// TIA Portal project "LECTOR CODIGO DE BARRAS" (V11)

(* hardware
DEVICE "S7300/ET200 station_1"  SIMATIC 300-Station
   slot 0: "Perfil soporte_0"  Rail  6ES7 390-1***0-0AA0
   slot 2: "PLC_1"  CPU 313C-2 DP  6ES7 313-6CF03-0AB0  V2.6
      slot 0: "Interfaz MPI_1"  MPI
      slot 1: "Interfaz DP_1"  DP
      slot 2: "DI16/DO16_1"  DI16/DO16
      slot 4: "Contaje_1"  Counter
   slot 4: "CP 343-1 Lean_1"  CP 343-1 LEAN  6GK7 343-1CX10-0XE0  V2.4
*)

// ===== PLC "PLC_1"  CPU 313C-2 DP =====

VAR_GLOBAL   // PLC tag table "Tabla de variables estándar"
   "ON PERMITE OFF NO" AT %I0.0 : Bool;
   "CANCELA LECTURA" AT %I0.1 : Bool;
   "Tag_2" AT %M0.0 : Bool;
   "Tag_4" AT %M0.1 : Bool;
   "Tag_5" AT %MW6 : Int;
   "Tag_7" AT %MW8 : Word;
   "Tag_1" AT %MW10 : Int;
   "Tag_3" AT %MD12 : Real;
   "Tag_6" AT %MW16 : Int;
   "Tag_14" AT %MD18 : Real;
   "Tag_15" AT %MW22 : Int;
   "Tag_16" AT %MD24 : Real;
   "Tag_17" AT %MW28 : Int;
   "Tag_18" AT %MD30 : Real;
   "Tag_19" AT %MD34 : Real;
   "Tag_20" AT %MD40 : Real;
   "RECTIFICAR FACTURA" AT %I0.2 : Bool;
   "RESET" AT %I0.3 : Bool;
   "Tag_8" AT %I0.4 : Bool;
   "Tag_9" AT %I0.5 : Bool;
   "Tag_10" AT %I0.6 : Bool;
   "Tag_11" AT %I0.7 : Bool;
   "Tag_12" AT %I1.0 : Bool;
   "Tag_13" AT %I1.1 : Bool;
   "Tag_21" AT %I1.2 : Bool;
   "Tag_22" AT %I1.3 : Bool;
   "Tag_23" AT %I1.4 : Bool;
   "Tag_24" AT %I1.5 : Bool;
   "Tag_25" AT %Q0.0 : Bool;
   "Tag_26" AT %Q0.1 : Bool;
   "Tag_27" AT %Q0.2 : Bool;
   "Tag_28" AT %Q0.3 : Bool;
   "Tag_29" AT %Q0.4 : Bool;
   "Tag_30" AT %I1.6 : Bool;
END_VAR

DATA_BLOCK "CODIGO CAMEL"   // DB1
{ S7_Optimized_Access := 'FALSE' }
VERSION : 0.1
   VAR
      CAMEL : Array [0..20] of Byte;
   END_VAR
BEGIN
   CAMEL[0] := '8';
   CAMEL[1] := '4';
   CAMEL[2] := '1';
   CAMEL[3] := '6';
   CAMEL[4] := '5';
   CAMEL[5] := '9';
   CAMEL[6] := '6';
   CAMEL[7] := '1';
END_DATA_BLOCK

DATA_BLOCK "CODIGO PALL MALL"   // DB2
{ S7_Optimized_Access := 'FALSE' }
VERSION : 0.1
   VAR
      "PALL MALL" : Array [0..20] of Byte;
   END_VAR
BEGIN
   "PALL MALL"[0] := '8';
   "PALL MALL"[1] := '4';
   "PALL MALL"[2] := '1';
   "PALL MALL"[3] := '6';
   "PALL MALL"[4] := '0';
   "PALL MALL"[5] := '9';
   "PALL MALL"[6] := '6';
   "PALL MALL"[7] := '6';
END_DATA_BLOCK

DATA_BLOCK "CODIGO FORTUNA"   // DB3
{ S7_Optimized_Access := 'FALSE' }
VERSION : 0.1
   VAR
      FORTUNA : Array [0..20] of Byte;
   END_VAR
BEGIN
   FORTUNA[0] := '8';
   FORTUNA[1] := '4';
   FORTUNA[2] := '1';
   FORTUNA[3] := '6';
   FORTUNA[4] := '0';
   FORTUNA[5] := '0';
   FORTUNA[6] := '2';
   FORTUNA[7] := '7';
END_DATA_BLOCK

DATA_BLOCK "LECTURA LECTOR"   // DB4
{ S7_Optimized_Access := 'FALSE' }
VERSION : 0.1
   VAR
      "LECTURA LECTOR" : Array [0..20] of Byte;
   END_VAR
BEGIN
END_DATA_BLOCK

DATA_BLOCK "CODIGO LUCKY"   // DB6
{ S7_Optimized_Access := 'FALSE' }
VERSION : 0.1
   VAR
      "CODIGO LUCKY" : Array [0..20] of Byte;
   END_VAR
BEGIN
   "CODIGO LUCKY"[0] := '8';
   "CODIGO LUCKY"[1] := '4';
   "CODIGO LUCKY"[2] := '1';
   "CODIGO LUCKY"[3] := '6';
   "CODIGO LUCKY"[4] := '0';
   "CODIGO LUCKY"[5] := '0';
   "CODIGO LUCKY"[6] := '8';
   "CODIGO LUCKY"[7] := '9';
END_DATA_BLOCK

DATA_BLOCK "DATOS AUXILIARES"   // DB7
{ S7_Optimized_Access := 'FALSE' }
VERSION : 0.1
   VAR
      DATOS : Array [0..41] of Bool;
      "CONTADOR UNID." : Array [0..3] of Int;
      "CONTADOR PVP TOTAL" : Array [0..3] of Real;
      "CONTADOR FACTURA TOTAL" : Array [0..0] of Real;
      "BOBINAS AUX." : Array [0..8] of Bool;
   END_VAR
BEGIN
END_DATA_BLOCK

FUNCTION "REGISTRO PALL MALL." : Void   // FC1, LAD
{ S7_Optimized_Access := 'FALSE' }
VERSION : 0.1
   VAR_OUTPUT
      "UNIDADES PALL MALL" : Int;
      "P.V.P. TOTAL" : Real;
   END_VAR
   VAR_TEMP   // added for the SCL form of the ladder/FBD networks
      _w1 : Bool;
      _w2 : Bool;
   END_VAR
BEGIN

REGION Network 1
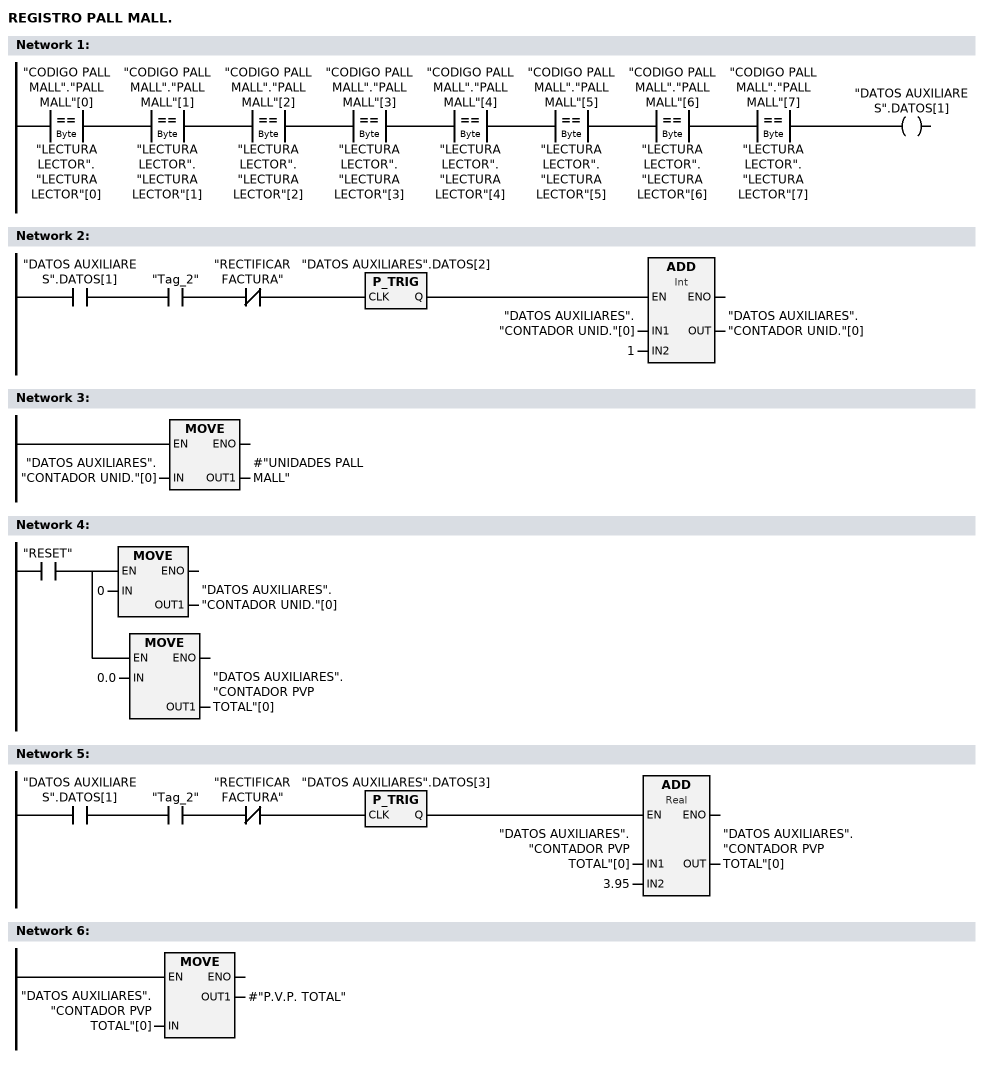
   RUNG wire#powerrail
      { S7_Templates := "SrcType := Byte" } EQ_Contact(in1 := "CODIGO PALL MALL"."PALL MALL"[0], in2 := "LECTURA LECTOR"."LECTURA LECTOR"[0])
      { S7_Templates := "SrcType := Byte" } EQ_Contact(in1 := "CODIGO PALL MALL"."PALL MALL"[1], in2 := "LECTURA LECTOR"."LECTURA LECTOR"[1])
      { S7_Templates := "SrcType := Byte" } EQ_Contact(in1 := "CODIGO PALL MALL"."PALL MALL"[2], in2 := "LECTURA LECTOR"."LECTURA LECTOR"[2])
      { S7_Templates := "SrcType := Byte" } EQ_Contact(in1 := "CODIGO PALL MALL"."PALL MALL"[3], in2 := "LECTURA LECTOR"."LECTURA LECTOR"[3])
      { S7_Templates := "SrcType := Byte" } EQ_Contact(in1 := "CODIGO PALL MALL"."PALL MALL"[4], in2 := "LECTURA LECTOR"."LECTURA LECTOR"[4])
      { S7_Templates := "SrcType := Byte" } EQ_Contact(in1 := "CODIGO PALL MALL"."PALL MALL"[5], in2 := "LECTURA LECTOR"."LECTURA LECTOR"[5])
      { S7_Templates := "SrcType := Byte" } EQ_Contact(in1 := "CODIGO PALL MALL"."PALL MALL"[6], in2 := "LECTURA LECTOR"."LECTURA LECTOR"[6])
      { S7_Templates := "SrcType := Byte" } EQ_Contact(in1 := "CODIGO PALL MALL"."PALL MALL"[7], in2 := "LECTURA LECTOR"."LECTURA LECTOR"[7])
      Coil( "DATOS AUXILIARES".DATOS[1] )
   END_RUNG
   // the same network as SCL:
   "DATOS AUXILIARES".DATOS[1] := ("CODIGO PALL MALL"."PALL MALL"[0] = "LECTURA LECTOR"."LECTURA LECTOR"[0]) AND ("CODIGO PALL MALL"."PALL MALL"[1] = "LECTURA LECTOR"."LECTURA LECTOR"[1]) AND ("CODIGO PALL MALL"."PALL MALL"[2] = "LECTURA LECTOR"."LECTURA LECTOR"[2]) AND ("CODIGO PALL MALL"."PALL MALL"[3] = "LECTURA LECTOR"."LECTURA LECTOR"[3]) AND ("CODIGO PALL MALL"."PALL MALL"[4] = "LECTURA LECTOR"."LECTURA LECTOR"[4]) AND ("CODIGO PALL MALL"."PALL MALL"[5] = "LECTURA LECTOR"."LECTURA LECTOR"[5]) AND ("CODIGO PALL MALL"."PALL MALL"[6] = "LECTURA LECTOR"."LECTURA LECTOR"[6]) AND ("CODIGO PALL MALL"."PALL MALL"[7] = "LECTURA LECTOR"."LECTURA LECTOR"[7]);
END_REGION

REGION Network 2
   RUNG wire#powerrail
      Contact( "DATOS AUXILIARES".DATOS[1] )
      Contact( "Tag_2" )
      I_Contact( "RECTIFICAR FACTURA" )
      P_Trig( "DATOS AUXILIARES".DATOS[2] )
      { S7_Templates := "SrcType := Int"; S7_GenerateENO := "TRUE" } Add(in1 := "DATOS AUXILIARES"."CONTADOR UNID."[0], in2 := 1, out => "DATOS AUXILIARES"."CONTADOR UNID."[0])
   END_RUNG
   // the same network as SCL:
   #_w1 := "DATOS AUXILIARES".DATOS[1] AND "Tag_2" AND NOT "RECTIFICAR FACTURA";
   #_w2 := #_w1 AND NOT "DATOS AUXILIARES".DATOS[2];   // rising edge
   "DATOS AUXILIARES".DATOS[2] := #_w1;
   IF #_w2 THEN "DATOS AUXILIARES"."CONTADOR UNID."[0] := "DATOS AUXILIARES"."CONTADOR UNID."[0] + 1; END_IF;
END_REGION

REGION Network 3
   RUNG wire#powerrail
      { S7_GenerateENO := "TRUE" } Move(in := "DATOS AUXILIARES"."CONTADOR UNID."[0], out1 => #"UNIDADES PALL MALL")
   END_RUNG
   // the same network as SCL:
   #"UNIDADES PALL MALL" := "DATOS AUXILIARES"."CONTADOR UNID."[0];
END_REGION

REGION Network 4
   RUNG wire#powerrail
      Contact( "RESET" )
      wire#w1
      { S7_GenerateENO := "TRUE" } Move(in := 0, out1 => "DATOS AUXILIARES"."CONTADOR UNID."[0])
   END_RUNG
   RUNG wire#w1
      { S7_GenerateENO := "TRUE" } Move(in := 0.0, out1 => "DATOS AUXILIARES"."CONTADOR PVP TOTAL"[0])
   END_RUNG
   // the same network as SCL:
   IF "RESET" THEN
       "DATOS AUXILIARES"."CONTADOR UNID."[0] := 0;
       "DATOS AUXILIARES"."CONTADOR PVP TOTAL"[0] := 0.0;
   END_IF;
END_REGION

REGION Network 5
   RUNG wire#powerrail
      Contact( "DATOS AUXILIARES".DATOS[1] )
      Contact( "Tag_2" )
      I_Contact( "RECTIFICAR FACTURA" )
      P_Trig( "DATOS AUXILIARES".DATOS[3] )
      { S7_Templates := "SrcType := Real"; S7_GenerateENO := "TRUE" } Add(in1 := "DATOS AUXILIARES"."CONTADOR PVP TOTAL"[0], in2 := 3.95, out => "DATOS AUXILIARES"."CONTADOR PVP TOTAL"[0])
   END_RUNG
   // the same network as SCL:
   #_w1 := "DATOS AUXILIARES".DATOS[1] AND "Tag_2" AND NOT "RECTIFICAR FACTURA";
   #_w2 := #_w1 AND NOT "DATOS AUXILIARES".DATOS[3];   // rising edge
   "DATOS AUXILIARES".DATOS[3] := #_w1;
   IF #_w2 THEN
       "DATOS AUXILIARES"."CONTADOR PVP TOTAL"[0] := "DATOS AUXILIARES"."CONTADOR PVP TOTAL"[0] + 3.95;
   END_IF;
END_REGION

REGION Network 6
   RUNG wire#powerrail
      { S7_GenerateENO := "TRUE" } Move(in := "DATOS AUXILIARES"."CONTADOR PVP TOTAL"[0], out1 => #"P.V.P. TOTAL")
   END_RUNG
   // the same network as SCL:
   #"P.V.P. TOTAL" := "DATOS AUXILIARES"."CONTADOR PVP TOTAL"[0];
END_REGION
END_FUNCTION

FUNCTION "REGISTRO CAMELL" : Void   // FC2, LAD
{ S7_Optimized_Access := 'FALSE' }
VERSION : 0.1
   VAR_OUTPUT
      "UNIDADES CAMELL" : Int;
      "PVP TOTAL" : Real;
   END_VAR
   VAR_TEMP   // added for the SCL form of the ladder/FBD networks
      _w1 : Bool;
      _w2 : Bool;
   END_VAR
BEGIN

REGION Network 1
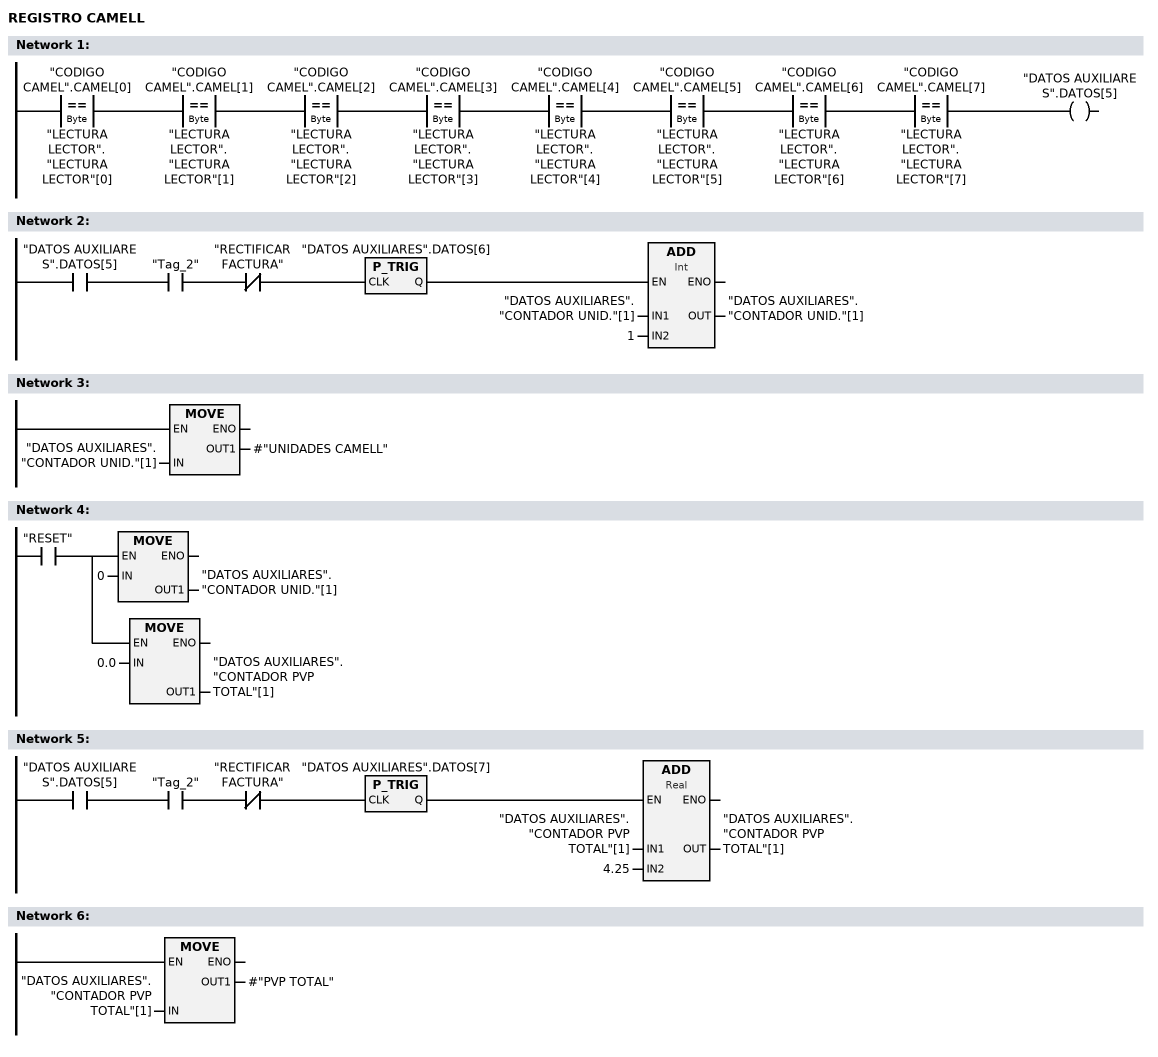
   RUNG wire#powerrail
      { S7_Templates := "SrcType := Byte" } EQ_Contact(in1 := "CODIGO CAMEL".CAMEL[0], in2 := "LECTURA LECTOR"."LECTURA LECTOR"[0])
      { S7_Templates := "SrcType := Byte" } EQ_Contact(in1 := "CODIGO CAMEL".CAMEL[1], in2 := "LECTURA LECTOR"."LECTURA LECTOR"[1])
      { S7_Templates := "SrcType := Byte" } EQ_Contact(in1 := "CODIGO CAMEL".CAMEL[2], in2 := "LECTURA LECTOR"."LECTURA LECTOR"[2])
      { S7_Templates := "SrcType := Byte" } EQ_Contact(in1 := "CODIGO CAMEL".CAMEL[3], in2 := "LECTURA LECTOR"."LECTURA LECTOR"[3])
      { S7_Templates := "SrcType := Byte" } EQ_Contact(in1 := "CODIGO CAMEL".CAMEL[4], in2 := "LECTURA LECTOR"."LECTURA LECTOR"[4])
      { S7_Templates := "SrcType := Byte" } EQ_Contact(in1 := "CODIGO CAMEL".CAMEL[5], in2 := "LECTURA LECTOR"."LECTURA LECTOR"[5])
      { S7_Templates := "SrcType := Byte" } EQ_Contact(in1 := "CODIGO CAMEL".CAMEL[6], in2 := "LECTURA LECTOR"."LECTURA LECTOR"[6])
      { S7_Templates := "SrcType := Byte" } EQ_Contact(in1 := "CODIGO CAMEL".CAMEL[7], in2 := "LECTURA LECTOR"."LECTURA LECTOR"[7])
      Coil( "DATOS AUXILIARES".DATOS[5] )
   END_RUNG
   // the same network as SCL:
   "DATOS AUXILIARES".DATOS[5] := ("CODIGO CAMEL".CAMEL[0] = "LECTURA LECTOR"."LECTURA LECTOR"[0]) AND ("CODIGO CAMEL".CAMEL[1] = "LECTURA LECTOR"."LECTURA LECTOR"[1]) AND ("CODIGO CAMEL".CAMEL[2] = "LECTURA LECTOR"."LECTURA LECTOR"[2]) AND ("CODIGO CAMEL".CAMEL[3] = "LECTURA LECTOR"."LECTURA LECTOR"[3]) AND ("CODIGO CAMEL".CAMEL[4] = "LECTURA LECTOR"."LECTURA LECTOR"[4]) AND ("CODIGO CAMEL".CAMEL[5] = "LECTURA LECTOR"."LECTURA LECTOR"[5]) AND ("CODIGO CAMEL".CAMEL[6] = "LECTURA LECTOR"."LECTURA LECTOR"[6]) AND ("CODIGO CAMEL".CAMEL[7] = "LECTURA LECTOR"."LECTURA LECTOR"[7]);
END_REGION

REGION Network 2
   RUNG wire#powerrail
      Contact( "DATOS AUXILIARES".DATOS[5] )
      Contact( "Tag_2" )
      I_Contact( "RECTIFICAR FACTURA" )
      P_Trig( "DATOS AUXILIARES".DATOS[6] )
      { S7_Templates := "SrcType := Int"; S7_GenerateENO := "TRUE" } Add(in1 := "DATOS AUXILIARES"."CONTADOR UNID."[1], in2 := 1, out => "DATOS AUXILIARES"."CONTADOR UNID."[1])
   END_RUNG
   // the same network as SCL:
   #_w1 := "DATOS AUXILIARES".DATOS[5] AND "Tag_2" AND NOT "RECTIFICAR FACTURA";
   #_w2 := #_w1 AND NOT "DATOS AUXILIARES".DATOS[6];   // rising edge
   "DATOS AUXILIARES".DATOS[6] := #_w1;
   IF #_w2 THEN "DATOS AUXILIARES"."CONTADOR UNID."[1] := "DATOS AUXILIARES"."CONTADOR UNID."[1] + 1; END_IF;
END_REGION

REGION Network 3
   RUNG wire#powerrail
      { S7_GenerateENO := "TRUE" } Move(in := "DATOS AUXILIARES"."CONTADOR UNID."[1], out1 => #"UNIDADES CAMELL")
   END_RUNG
   // the same network as SCL:
   #"UNIDADES CAMELL" := "DATOS AUXILIARES"."CONTADOR UNID."[1];
END_REGION

REGION Network 4
   RUNG wire#powerrail
      Contact( "RESET" )
      wire#w1
      { S7_GenerateENO := "TRUE" } Move(in := 0, out1 => "DATOS AUXILIARES"."CONTADOR UNID."[1])
   END_RUNG
   RUNG wire#w1
      { S7_GenerateENO := "TRUE" } Move(in := 0.0, out1 => "DATOS AUXILIARES"."CONTADOR PVP TOTAL"[1])
   END_RUNG
   // the same network as SCL:
   IF "RESET" THEN
       "DATOS AUXILIARES"."CONTADOR UNID."[1] := 0;
       "DATOS AUXILIARES"."CONTADOR PVP TOTAL"[1] := 0.0;
   END_IF;
END_REGION

REGION Network 5
   RUNG wire#powerrail
      Contact( "DATOS AUXILIARES".DATOS[5] )
      Contact( "Tag_2" )
      I_Contact( "RECTIFICAR FACTURA" )
      P_Trig( "DATOS AUXILIARES".DATOS[7] )
      { S7_Templates := "SrcType := Real"; S7_GenerateENO := "TRUE" } Add(in1 := "DATOS AUXILIARES"."CONTADOR PVP TOTAL"[1], in2 := 4.25, out => "DATOS AUXILIARES"."CONTADOR PVP TOTAL"[1])
   END_RUNG
   // the same network as SCL:
   #_w1 := "DATOS AUXILIARES".DATOS[5] AND "Tag_2" AND NOT "RECTIFICAR FACTURA";
   #_w2 := #_w1 AND NOT "DATOS AUXILIARES".DATOS[7];   // rising edge
   "DATOS AUXILIARES".DATOS[7] := #_w1;
   IF #_w2 THEN
       "DATOS AUXILIARES"."CONTADOR PVP TOTAL"[1] := "DATOS AUXILIARES"."CONTADOR PVP TOTAL"[1] + 4.25;
   END_IF;
END_REGION

REGION Network 6
   RUNG wire#powerrail
      { S7_GenerateENO := "TRUE" } Move(in := "DATOS AUXILIARES"."CONTADOR PVP TOTAL"[1], out1 => #"PVP TOTAL")
   END_RUNG
   // the same network as SCL:
   #"PVP TOTAL" := "DATOS AUXILIARES"."CONTADOR PVP TOTAL"[1];
END_REGION
END_FUNCTION

FUNCTION "REGISTRO FORTUNA" : Void   // FC3, LAD
{ S7_Optimized_Access := 'FALSE' }
VERSION : 0.1
   VAR_OUTPUT
      "UNIDADES FORTUNA" : Int;
      "PVP TOTAL" : Real;
   END_VAR
   VAR_TEMP   // added for the SCL form of the ladder/FBD networks
      _w1 : Bool;
      _w2 : Bool;
   END_VAR
BEGIN

REGION Network 1
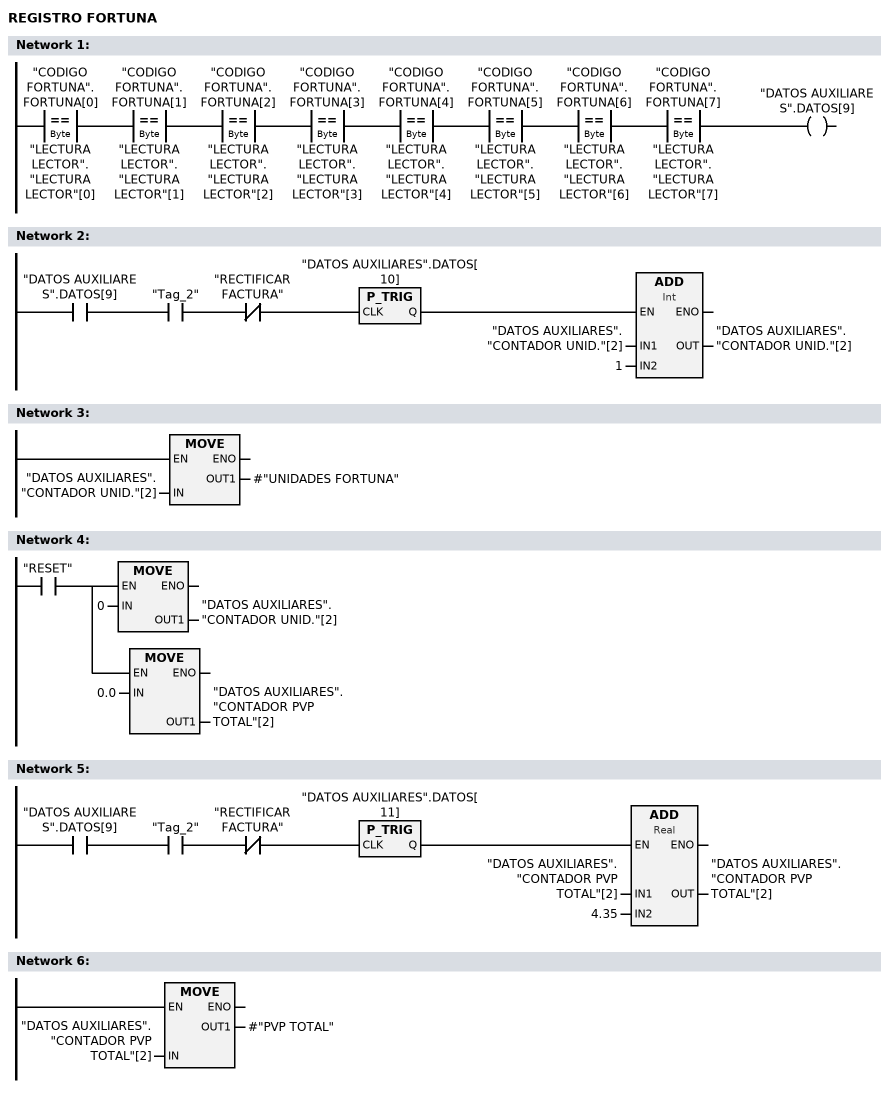
   RUNG wire#powerrail
      { S7_Templates := "SrcType := Byte" } EQ_Contact(in1 := "CODIGO FORTUNA".FORTUNA[0], in2 := "LECTURA LECTOR"."LECTURA LECTOR"[0])
      { S7_Templates := "SrcType := Byte" } EQ_Contact(in1 := "CODIGO FORTUNA".FORTUNA[1], in2 := "LECTURA LECTOR"."LECTURA LECTOR"[1])
      { S7_Templates := "SrcType := Byte" } EQ_Contact(in1 := "CODIGO FORTUNA".FORTUNA[2], in2 := "LECTURA LECTOR"."LECTURA LECTOR"[2])
      { S7_Templates := "SrcType := Byte" } EQ_Contact(in1 := "CODIGO FORTUNA".FORTUNA[3], in2 := "LECTURA LECTOR"."LECTURA LECTOR"[3])
      { S7_Templates := "SrcType := Byte" } EQ_Contact(in1 := "CODIGO FORTUNA".FORTUNA[4], in2 := "LECTURA LECTOR"."LECTURA LECTOR"[4])
      { S7_Templates := "SrcType := Byte" } EQ_Contact(in1 := "CODIGO FORTUNA".FORTUNA[5], in2 := "LECTURA LECTOR"."LECTURA LECTOR"[5])
      { S7_Templates := "SrcType := Byte" } EQ_Contact(in1 := "CODIGO FORTUNA".FORTUNA[6], in2 := "LECTURA LECTOR"."LECTURA LECTOR"[6])
      { S7_Templates := "SrcType := Byte" } EQ_Contact(in1 := "CODIGO FORTUNA".FORTUNA[7], in2 := "LECTURA LECTOR"."LECTURA LECTOR"[7])
      Coil( "DATOS AUXILIARES".DATOS[9] )
   END_RUNG
   // the same network as SCL:
   "DATOS AUXILIARES".DATOS[9] := ("CODIGO FORTUNA".FORTUNA[0] = "LECTURA LECTOR"."LECTURA LECTOR"[0]) AND ("CODIGO FORTUNA".FORTUNA[1] = "LECTURA LECTOR"."LECTURA LECTOR"[1]) AND ("CODIGO FORTUNA".FORTUNA[2] = "LECTURA LECTOR"."LECTURA LECTOR"[2]) AND ("CODIGO FORTUNA".FORTUNA[3] = "LECTURA LECTOR"."LECTURA LECTOR"[3]) AND ("CODIGO FORTUNA".FORTUNA[4] = "LECTURA LECTOR"."LECTURA LECTOR"[4]) AND ("CODIGO FORTUNA".FORTUNA[5] = "LECTURA LECTOR"."LECTURA LECTOR"[5]) AND ("CODIGO FORTUNA".FORTUNA[6] = "LECTURA LECTOR"."LECTURA LECTOR"[6]) AND ("CODIGO FORTUNA".FORTUNA[7] = "LECTURA LECTOR"."LECTURA LECTOR"[7]);
END_REGION

REGION Network 2
   RUNG wire#powerrail
      Contact( "DATOS AUXILIARES".DATOS[9] )
      Contact( "Tag_2" )
      I_Contact( "RECTIFICAR FACTURA" )
      P_Trig( "DATOS AUXILIARES".DATOS[10] )
      { S7_Templates := "SrcType := Int"; S7_GenerateENO := "TRUE" } Add(in1 := "DATOS AUXILIARES"."CONTADOR UNID."[2], in2 := 1, out => "DATOS AUXILIARES"."CONTADOR UNID."[2])
   END_RUNG
   // the same network as SCL:
   #_w1 := "DATOS AUXILIARES".DATOS[9] AND "Tag_2" AND NOT "RECTIFICAR FACTURA";
   #_w2 := #_w1 AND NOT "DATOS AUXILIARES".DATOS[10];   // rising edge
   "DATOS AUXILIARES".DATOS[10] := #_w1;
   IF #_w2 THEN "DATOS AUXILIARES"."CONTADOR UNID."[2] := "DATOS AUXILIARES"."CONTADOR UNID."[2] + 1; END_IF;
END_REGION

REGION Network 3
   RUNG wire#powerrail
      { S7_GenerateENO := "TRUE" } Move(in := "DATOS AUXILIARES"."CONTADOR UNID."[2], out1 => #"UNIDADES FORTUNA")
   END_RUNG
   // the same network as SCL:
   #"UNIDADES FORTUNA" := "DATOS AUXILIARES"."CONTADOR UNID."[2];
END_REGION

REGION Network 4
   RUNG wire#powerrail
      Contact( "RESET" )
      wire#w1
      { S7_GenerateENO := "TRUE" } Move(in := 0, out1 => "DATOS AUXILIARES"."CONTADOR UNID."[2])
   END_RUNG
   RUNG wire#w1
      { S7_GenerateENO := "TRUE" } Move(in := 0.0, out1 => "DATOS AUXILIARES"."CONTADOR PVP TOTAL"[2])
   END_RUNG
   // the same network as SCL:
   IF "RESET" THEN
       "DATOS AUXILIARES"."CONTADOR UNID."[2] := 0;
       "DATOS AUXILIARES"."CONTADOR PVP TOTAL"[2] := 0.0;
   END_IF;
END_REGION

REGION Network 5
   RUNG wire#powerrail
      Contact( "DATOS AUXILIARES".DATOS[9] )
      Contact( "Tag_2" )
      I_Contact( "RECTIFICAR FACTURA" )
      P_Trig( "DATOS AUXILIARES".DATOS[11] )
      { S7_Templates := "SrcType := Real"; S7_GenerateENO := "TRUE" } Add(in1 := "DATOS AUXILIARES"."CONTADOR PVP TOTAL"[2], in2 := 4.35, out => "DATOS AUXILIARES"."CONTADOR PVP TOTAL"[2])
   END_RUNG
   // the same network as SCL:
   #_w1 := "DATOS AUXILIARES".DATOS[9] AND "Tag_2" AND NOT "RECTIFICAR FACTURA";
   #_w2 := #_w1 AND NOT "DATOS AUXILIARES".DATOS[11];   // rising edge
   "DATOS AUXILIARES".DATOS[11] := #_w1;
   IF #_w2 THEN
       "DATOS AUXILIARES"."CONTADOR PVP TOTAL"[2] := "DATOS AUXILIARES"."CONTADOR PVP TOTAL"[2] + 4.35;
   END_IF;
END_REGION

REGION Network 6
   RUNG wire#powerrail
      { S7_GenerateENO := "TRUE" } Move(in := "DATOS AUXILIARES"."CONTADOR PVP TOTAL"[2], out1 => #"PVP TOTAL")
   END_RUNG
   // the same network as SCL:
   #"PVP TOTAL" := "DATOS AUXILIARES"."CONTADOR PVP TOTAL"[2];
END_REGION
END_FUNCTION

FUNCTION "REGISTRO LUCKY" : Void   // FC4, LAD
{ S7_Optimized_Access := 'FALSE' }
VERSION : 0.1
   VAR_OUTPUT
      "UNIDEDES LUCKY" : Int;
      "PVP TOTAL" : Real;
   END_VAR
   VAR_TEMP   // added for the SCL form of the ladder/FBD networks
      _w1 : Bool;
      _w2 : Bool;
   END_VAR
BEGIN

REGION Network 1
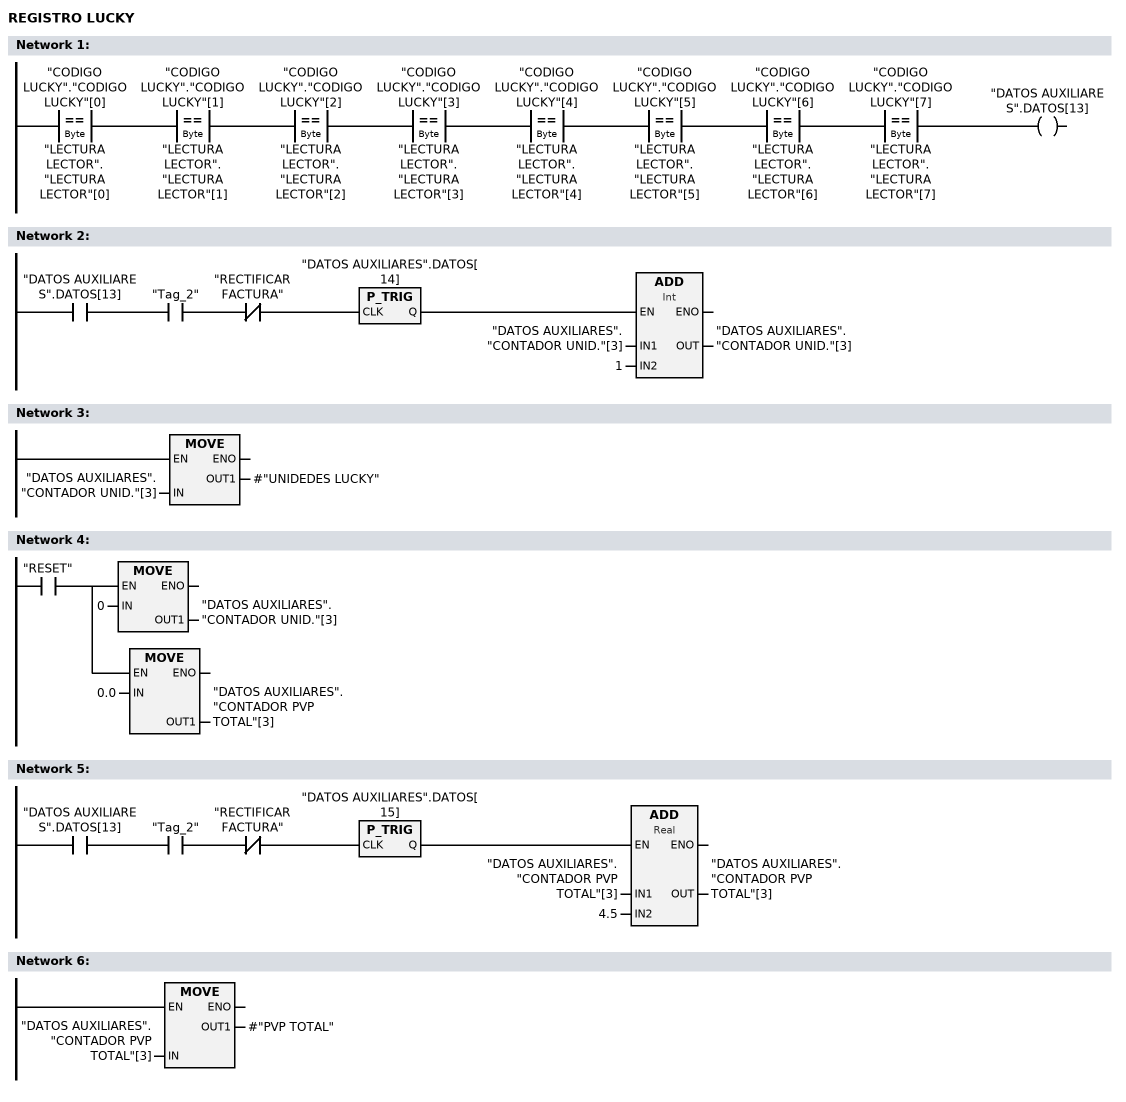
   RUNG wire#powerrail
      { S7_Templates := "SrcType := Byte" } EQ_Contact(in1 := "CODIGO LUCKY"."CODIGO LUCKY"[0], in2 := "LECTURA LECTOR"."LECTURA LECTOR"[0])
      { S7_Templates := "SrcType := Byte" } EQ_Contact(in1 := "CODIGO LUCKY"."CODIGO LUCKY"[1], in2 := "LECTURA LECTOR"."LECTURA LECTOR"[1])
      { S7_Templates := "SrcType := Byte" } EQ_Contact(in1 := "CODIGO LUCKY"."CODIGO LUCKY"[2], in2 := "LECTURA LECTOR"."LECTURA LECTOR"[2])
      { S7_Templates := "SrcType := Byte" } EQ_Contact(in1 := "CODIGO LUCKY"."CODIGO LUCKY"[3], in2 := "LECTURA LECTOR"."LECTURA LECTOR"[3])
      { S7_Templates := "SrcType := Byte" } EQ_Contact(in1 := "CODIGO LUCKY"."CODIGO LUCKY"[4], in2 := "LECTURA LECTOR"."LECTURA LECTOR"[4])
      { S7_Templates := "SrcType := Byte" } EQ_Contact(in1 := "CODIGO LUCKY"."CODIGO LUCKY"[5], in2 := "LECTURA LECTOR"."LECTURA LECTOR"[5])
      { S7_Templates := "SrcType := Byte" } EQ_Contact(in1 := "CODIGO LUCKY"."CODIGO LUCKY"[6], in2 := "LECTURA LECTOR"."LECTURA LECTOR"[6])
      { S7_Templates := "SrcType := Byte" } EQ_Contact(in1 := "CODIGO LUCKY"."CODIGO LUCKY"[7], in2 := "LECTURA LECTOR"."LECTURA LECTOR"[7])
      Coil( "DATOS AUXILIARES".DATOS[13] )
   END_RUNG
   // the same network as SCL:
   "DATOS AUXILIARES".DATOS[13] := ("CODIGO LUCKY"."CODIGO LUCKY"[0] = "LECTURA LECTOR"."LECTURA LECTOR"[0]) AND ("CODIGO LUCKY"."CODIGO LUCKY"[1] = "LECTURA LECTOR"."LECTURA LECTOR"[1]) AND ("CODIGO LUCKY"."CODIGO LUCKY"[2] = "LECTURA LECTOR"."LECTURA LECTOR"[2]) AND ("CODIGO LUCKY"."CODIGO LUCKY"[3] = "LECTURA LECTOR"."LECTURA LECTOR"[3]) AND ("CODIGO LUCKY"."CODIGO LUCKY"[4] = "LECTURA LECTOR"."LECTURA LECTOR"[4]) AND ("CODIGO LUCKY"."CODIGO LUCKY"[5] = "LECTURA LECTOR"."LECTURA LECTOR"[5]) AND ("CODIGO LUCKY"."CODIGO LUCKY"[6] = "LECTURA LECTOR"."LECTURA LECTOR"[6]) AND ("CODIGO LUCKY"."CODIGO LUCKY"[7] = "LECTURA LECTOR"."LECTURA LECTOR"[7]);
END_REGION

REGION Network 2
   RUNG wire#powerrail
      Contact( "DATOS AUXILIARES".DATOS[13] )
      Contact( "Tag_2" )
      I_Contact( "RECTIFICAR FACTURA" )
      P_Trig( "DATOS AUXILIARES".DATOS[14] )
      { S7_Templates := "SrcType := Int"; S7_GenerateENO := "TRUE" } Add(in1 := "DATOS AUXILIARES"."CONTADOR UNID."[3], in2 := 1, out => "DATOS AUXILIARES"."CONTADOR UNID."[3])
   END_RUNG
   // the same network as SCL:
   #_w1 := "DATOS AUXILIARES".DATOS[13] AND "Tag_2" AND NOT "RECTIFICAR FACTURA";
   #_w2 := #_w1 AND NOT "DATOS AUXILIARES".DATOS[14];   // rising edge
   "DATOS AUXILIARES".DATOS[14] := #_w1;
   IF #_w2 THEN "DATOS AUXILIARES"."CONTADOR UNID."[3] := "DATOS AUXILIARES"."CONTADOR UNID."[3] + 1; END_IF;
END_REGION

REGION Network 3
   RUNG wire#powerrail
      { S7_GenerateENO := "TRUE" } Move(in := "DATOS AUXILIARES"."CONTADOR UNID."[3], out1 => #"UNIDEDES LUCKY")
   END_RUNG
   // the same network as SCL:
   #"UNIDEDES LUCKY" := "DATOS AUXILIARES"."CONTADOR UNID."[3];
END_REGION

REGION Network 4
   RUNG wire#powerrail
      Contact( "RESET" )
      wire#w1
      { S7_GenerateENO := "TRUE" } Move(in := 0, out1 => "DATOS AUXILIARES"."CONTADOR UNID."[3])
   END_RUNG
   RUNG wire#w1
      { S7_GenerateENO := "TRUE" } Move(in := 0.0, out1 => "DATOS AUXILIARES"."CONTADOR PVP TOTAL"[3])
   END_RUNG
   // the same network as SCL:
   IF "RESET" THEN
       "DATOS AUXILIARES"."CONTADOR UNID."[3] := 0;
       "DATOS AUXILIARES"."CONTADOR PVP TOTAL"[3] := 0.0;
   END_IF;
END_REGION

REGION Network 5
   RUNG wire#powerrail
      Contact( "DATOS AUXILIARES".DATOS[13] )
      Contact( "Tag_2" )
      I_Contact( "RECTIFICAR FACTURA" )
      P_Trig( "DATOS AUXILIARES".DATOS[15] )
      { S7_Templates := "SrcType := Real"; S7_GenerateENO := "TRUE" } Add(in1 := "DATOS AUXILIARES"."CONTADOR PVP TOTAL"[3], in2 := 4.5, out => "DATOS AUXILIARES"."CONTADOR PVP TOTAL"[3])
   END_RUNG
   // the same network as SCL:
   #_w1 := "DATOS AUXILIARES".DATOS[13] AND "Tag_2" AND NOT "RECTIFICAR FACTURA";
   #_w2 := #_w1 AND NOT "DATOS AUXILIARES".DATOS[15];   // rising edge
   "DATOS AUXILIARES".DATOS[15] := #_w1;
   IF #_w2 THEN
       "DATOS AUXILIARES"."CONTADOR PVP TOTAL"[3] := "DATOS AUXILIARES"."CONTADOR PVP TOTAL"[3] + 4.5;
   END_IF;
END_REGION

REGION Network 6
   RUNG wire#powerrail
      { S7_GenerateENO := "TRUE" } Move(in := "DATOS AUXILIARES"."CONTADOR PVP TOTAL"[3], out1 => #"PVP TOTAL")
   END_RUNG
   // the same network as SCL:
   #"PVP TOTAL" := "DATOS AUXILIARES"."CONTADOR PVP TOTAL"[3];
END_REGION
END_FUNCTION

FUNCTION "FACTURA TOTAL" : Void   // FC5, LAD
{ S7_Optimized_Access := 'FALSE' }
VERSION : 0.1
   VAR_OUTPUT
      "FATURA TOTAL" : Real;
   END_VAR
   VAR_TEMP   // added for the SCL form of the ladder/FBD networks
      _w1 : Bool;
      _w2 : Bool;
   END_VAR
BEGIN

REGION Network 1: SUMA PRECIO PALL MALL POR UNIDAD A CONTADOR FACTURA TOTAL
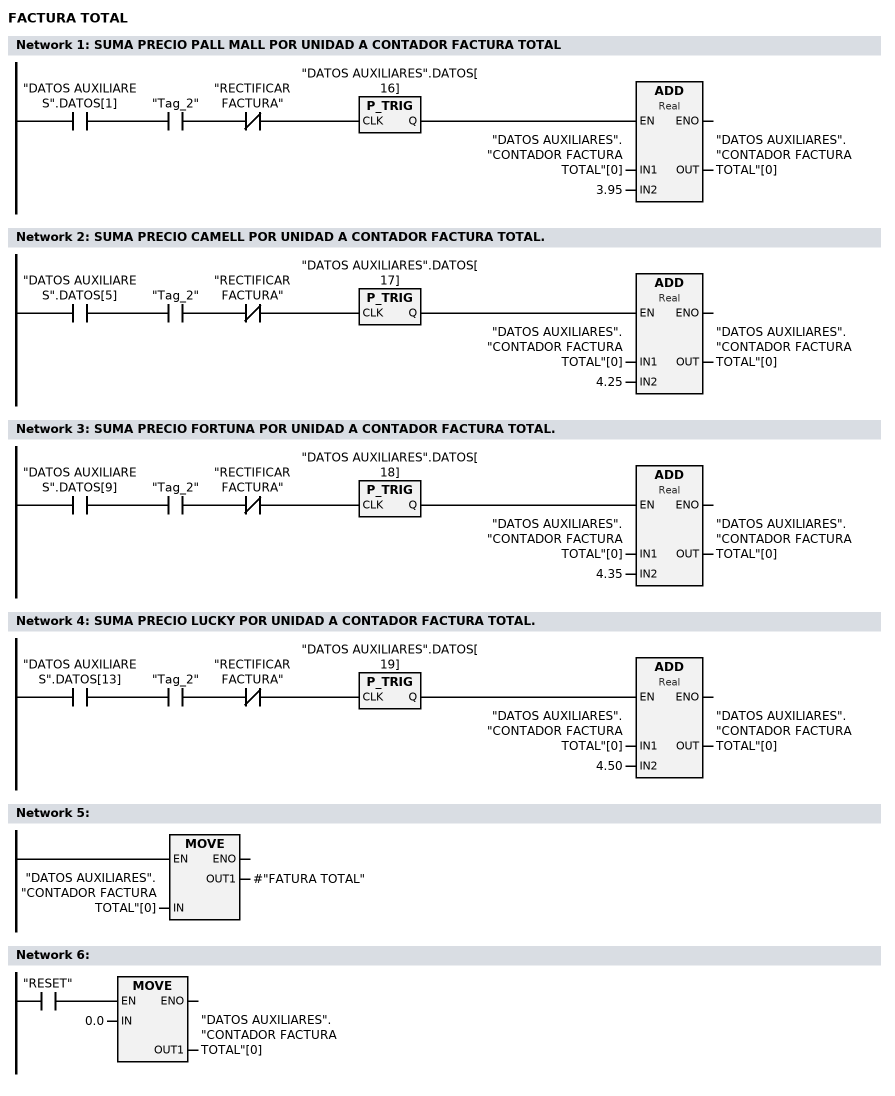
   RUNG wire#powerrail
      Contact( "DATOS AUXILIARES".DATOS[1] )
      Contact( "Tag_2" )
      I_Contact( "RECTIFICAR FACTURA" )
      P_Trig( "DATOS AUXILIARES".DATOS[16] )
      { S7_Templates := "SrcType := Real"; S7_GenerateENO := "TRUE" } Add(in1 := "DATOS AUXILIARES"."CONTADOR FACTURA TOTAL"[0], in2 := 3.95, out => "DATOS AUXILIARES"."CONTADOR FACTURA TOTAL"[0])
   END_RUNG
   // the same network as SCL:
   #_w1 := "DATOS AUXILIARES".DATOS[1] AND "Tag_2" AND NOT "RECTIFICAR FACTURA";
   #_w2 := #_w1 AND NOT "DATOS AUXILIARES".DATOS[16];   // rising edge
   "DATOS AUXILIARES".DATOS[16] := #_w1;
   IF #_w2 THEN
       "DATOS AUXILIARES"."CONTADOR FACTURA TOTAL"[0] := "DATOS AUXILIARES"."CONTADOR FACTURA TOTAL"[0] + 3.95;
   END_IF;
END_REGION

REGION Network 2: SUMA PRECIO CAMELL POR UNIDAD A CONTADOR FACTURA TOTAL.
   RUNG wire#powerrail
      Contact( "DATOS AUXILIARES".DATOS[5] )
      Contact( "Tag_2" )
      I_Contact( "RECTIFICAR FACTURA" )
      P_Trig( "DATOS AUXILIARES".DATOS[17] )
      { S7_Templates := "SrcType := Real"; S7_GenerateENO := "TRUE" } Add(in1 := "DATOS AUXILIARES"."CONTADOR FACTURA TOTAL"[0], in2 := 4.25, out => "DATOS AUXILIARES"."CONTADOR FACTURA TOTAL"[0])
   END_RUNG
   // the same network as SCL:
   #_w1 := "DATOS AUXILIARES".DATOS[5] AND "Tag_2" AND NOT "RECTIFICAR FACTURA";
   #_w2 := #_w1 AND NOT "DATOS AUXILIARES".DATOS[17];   // rising edge
   "DATOS AUXILIARES".DATOS[17] := #_w1;
   IF #_w2 THEN
       "DATOS AUXILIARES"."CONTADOR FACTURA TOTAL"[0] := "DATOS AUXILIARES"."CONTADOR FACTURA TOTAL"[0] + 4.25;
   END_IF;
END_REGION

REGION Network 3: SUMA PRECIO FORTUNA POR UNIDAD A CONTADOR FACTURA TOTAL.
   RUNG wire#powerrail
      Contact( "DATOS AUXILIARES".DATOS[9] )
      Contact( "Tag_2" )
      I_Contact( "RECTIFICAR FACTURA" )
      P_Trig( "DATOS AUXILIARES".DATOS[18] )
      { S7_Templates := "SrcType := Real"; S7_GenerateENO := "TRUE" } Add(in1 := "DATOS AUXILIARES"."CONTADOR FACTURA TOTAL"[0], in2 := 4.35, out => "DATOS AUXILIARES"."CONTADOR FACTURA TOTAL"[0])
   END_RUNG
   // the same network as SCL:
   #_w1 := "DATOS AUXILIARES".DATOS[9] AND "Tag_2" AND NOT "RECTIFICAR FACTURA";
   #_w2 := #_w1 AND NOT "DATOS AUXILIARES".DATOS[18];   // rising edge
   "DATOS AUXILIARES".DATOS[18] := #_w1;
   IF #_w2 THEN
       "DATOS AUXILIARES"."CONTADOR FACTURA TOTAL"[0] := "DATOS AUXILIARES"."CONTADOR FACTURA TOTAL"[0] + 4.35;
   END_IF;
END_REGION

REGION Network 4: SUMA PRECIO LUCKY POR UNIDAD A CONTADOR FACTURA TOTAL.
   RUNG wire#powerrail
      Contact( "DATOS AUXILIARES".DATOS[13] )
      Contact( "Tag_2" )
      I_Contact( "RECTIFICAR FACTURA" )
      P_Trig( "DATOS AUXILIARES".DATOS[19] )
      { S7_Templates := "SrcType := Real"; S7_GenerateENO := "TRUE" } Add(in1 := "DATOS AUXILIARES"."CONTADOR FACTURA TOTAL"[0], in2 := 4.50, out => "DATOS AUXILIARES"."CONTADOR FACTURA TOTAL"[0])
   END_RUNG
   // the same network as SCL:
   #_w1 := "DATOS AUXILIARES".DATOS[13] AND "Tag_2" AND NOT "RECTIFICAR FACTURA";
   #_w2 := #_w1 AND NOT "DATOS AUXILIARES".DATOS[19];   // rising edge
   "DATOS AUXILIARES".DATOS[19] := #_w1;
   IF #_w2 THEN
       "DATOS AUXILIARES"."CONTADOR FACTURA TOTAL"[0] := "DATOS AUXILIARES"."CONTADOR FACTURA TOTAL"[0] + 4.50;
   END_IF;
END_REGION

REGION Network 5
   RUNG wire#powerrail
      { S7_GenerateENO := "TRUE" } Move(in := "DATOS AUXILIARES"."CONTADOR FACTURA TOTAL"[0], out1 => #"FATURA TOTAL")
   END_RUNG
   // the same network as SCL:
   #"FATURA TOTAL" := "DATOS AUXILIARES"."CONTADOR FACTURA TOTAL"[0];
END_REGION

REGION Network 6
   RUNG wire#powerrail
      Contact( "RESET" )
      { S7_GenerateENO := "TRUE" } Move(in := 0.0, out1 => "DATOS AUXILIARES"."CONTADOR FACTURA TOTAL"[0])
   END_RUNG
   // the same network as SCL:
   IF "RESET" THEN "DATOS AUXILIARES"."CONTADOR FACTURA TOTAL"[0] := 0.0; END_IF;
END_REGION
END_FUNCTION

FUNCTION "CONSULTAR PRECIO" : Void   // FC6, LAD
{ S7_Optimized_Access := 'FALSE' }
VERSION : 0.1
   VAR_OUTPUT
      "PVP PAQUETE" : Real;
   END_VAR
   VAR_TEMP   // added for the SCL form of the ladder/FBD networks
      _w1 : Bool;
      _w2 : Bool;
   END_VAR
BEGIN

REGION Network 1: PALL MALL
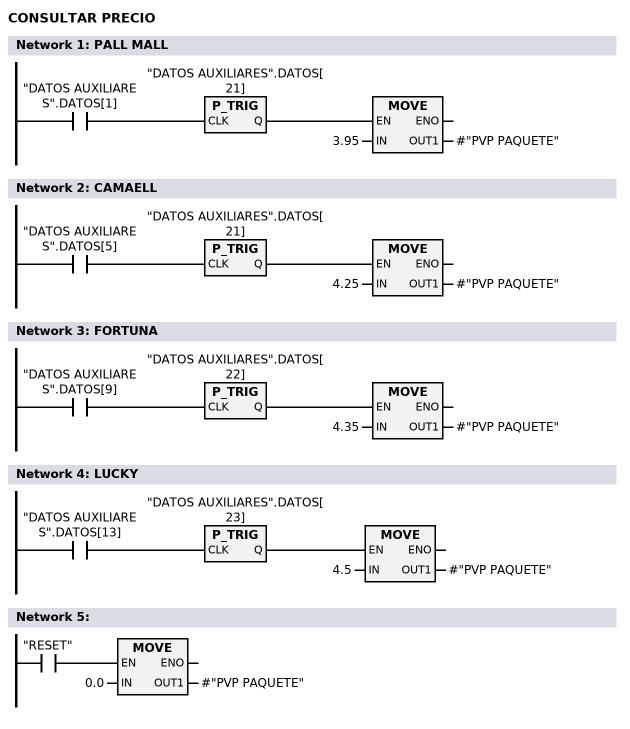
   RUNG wire#powerrail
      Contact( "DATOS AUXILIARES".DATOS[1] )
      P_Trig( "DATOS AUXILIARES".DATOS[21] )
      { S7_GenerateENO := "TRUE" } Move(in := 3.95, out1 => #"PVP PAQUETE")
   END_RUNG
   // the same network as SCL:
   #_w1 := "DATOS AUXILIARES".DATOS[1];
   #_w2 := #_w1 AND NOT "DATOS AUXILIARES".DATOS[21];   // rising edge
   "DATOS AUXILIARES".DATOS[21] := #_w1;
   IF #_w2 THEN #"PVP PAQUETE" := 3.95; END_IF;
END_REGION

REGION Network 2: CAMAELL
   RUNG wire#powerrail
      Contact( "DATOS AUXILIARES".DATOS[5] )
      P_Trig( "DATOS AUXILIARES".DATOS[21] )
      { S7_GenerateENO := "TRUE" } Move(in := 4.25, out1 => #"PVP PAQUETE")
   END_RUNG
   // the same network as SCL:
   #_w1 := "DATOS AUXILIARES".DATOS[5];
   #_w2 := #_w1 AND NOT "DATOS AUXILIARES".DATOS[21];   // rising edge
   "DATOS AUXILIARES".DATOS[21] := #_w1;
   IF #_w2 THEN #"PVP PAQUETE" := 4.25; END_IF;
END_REGION

REGION Network 3: FORTUNA
   RUNG wire#powerrail
      Contact( "DATOS AUXILIARES".DATOS[9] )
      P_Trig( "DATOS AUXILIARES".DATOS[22] )
      { S7_GenerateENO := "TRUE" } Move(in := 4.35, out1 => #"PVP PAQUETE")
   END_RUNG
   // the same network as SCL:
   #_w1 := "DATOS AUXILIARES".DATOS[9];
   #_w2 := #_w1 AND NOT "DATOS AUXILIARES".DATOS[22];   // rising edge
   "DATOS AUXILIARES".DATOS[22] := #_w1;
   IF #_w2 THEN #"PVP PAQUETE" := 4.35; END_IF;
END_REGION

REGION Network 4: LUCKY
   RUNG wire#powerrail
      Contact( "DATOS AUXILIARES".DATOS[13] )
      P_Trig( "DATOS AUXILIARES".DATOS[23] )
      { S7_GenerateENO := "TRUE" } Move(in := 4.5, out1 => #"PVP PAQUETE")
   END_RUNG
   // the same network as SCL:
   #_w1 := "DATOS AUXILIARES".DATOS[13];
   #_w2 := #_w1 AND NOT "DATOS AUXILIARES".DATOS[23];   // rising edge
   "DATOS AUXILIARES".DATOS[23] := #_w1;
   IF #_w2 THEN #"PVP PAQUETE" := 4.5; END_IF;
END_REGION

REGION Network 5
   RUNG wire#powerrail
      Contact( "RESET" )
      { S7_GenerateENO := "TRUE" } Move(in := 0.0, out1 => #"PVP PAQUETE")
   END_RUNG
   // the same network as SCL:
   IF "RESET" THEN #"PVP PAQUETE" := 0.0; END_IF;
END_REGION
END_FUNCTION

FUNCTION "RECTIFICACION FACTURA" : Void   // FC7, LAD
{ S7_Optimized_Access := 'FALSE' }
VERSION : 0.1
   VAR_INPUT
      RECTIFCAR : Bool;
   END_VAR
   VAR_TEMP   // added for the SCL form of the ladder/FBD networks
      _w1 : Bool;
      _w2 : Bool;
   END_VAR
BEGIN

REGION Network 1: RESTA PALL MALL
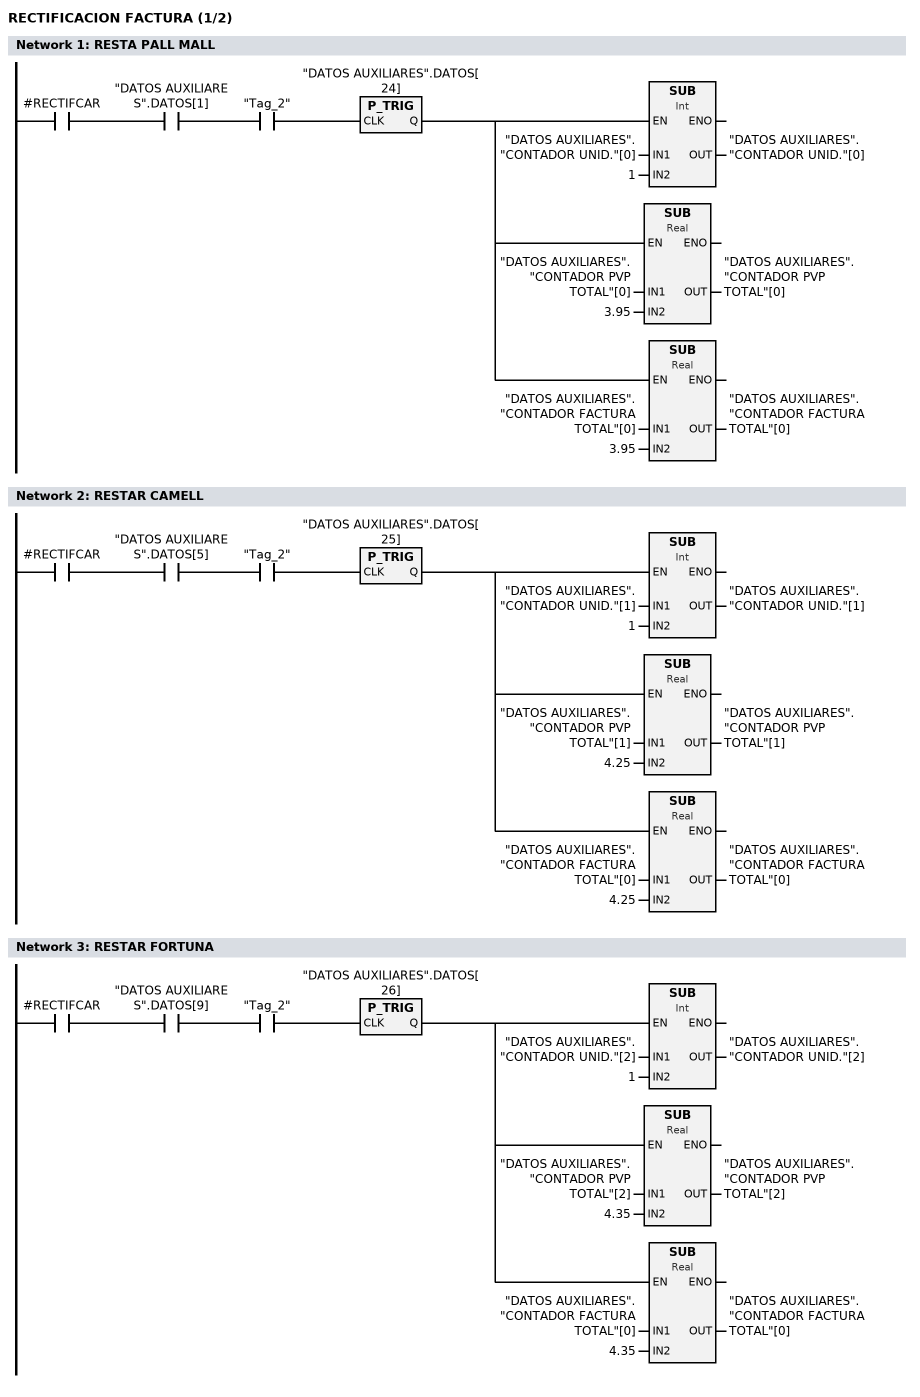
   RUNG wire#powerrail
      Contact( #RECTIFCAR )
      Contact( "DATOS AUXILIARES".DATOS[1] )
      Contact( "Tag_2" )
      P_Trig( "DATOS AUXILIARES".DATOS[24] )
      wire#w1
      { S7_Templates := "SrcType := Int"; S7_GenerateENO := "TRUE" } Sub(in1 := "DATOS AUXILIARES"."CONTADOR UNID."[0], in2 := 1, out => "DATOS AUXILIARES"."CONTADOR UNID."[0])
   END_RUNG
   RUNG wire#w1
      { S7_Templates := "SrcType := Real"; S7_GenerateENO := "TRUE" } Sub(in1 := "DATOS AUXILIARES"."CONTADOR PVP TOTAL"[0], in2 := 3.95, out => "DATOS AUXILIARES"."CONTADOR PVP TOTAL"[0])
   END_RUNG
   RUNG wire#w1
      { S7_Templates := "SrcType := Real"; S7_GenerateENO := "TRUE" } Sub(in1 := "DATOS AUXILIARES"."CONTADOR FACTURA TOTAL"[0], in2 := 3.95, out => "DATOS AUXILIARES"."CONTADOR FACTURA TOTAL"[0])
   END_RUNG
   // the same network as SCL:
   #_w1 := #RECTIFCAR AND "DATOS AUXILIARES".DATOS[1] AND "Tag_2";
   #_w2 := #_w1 AND NOT "DATOS AUXILIARES".DATOS[24];   // rising edge
   "DATOS AUXILIARES".DATOS[24] := #_w1;
   IF #_w2 THEN
       "DATOS AUXILIARES"."CONTADOR UNID."[0] := "DATOS AUXILIARES"."CONTADOR UNID."[0] - 1;
       "DATOS AUXILIARES"."CONTADOR PVP TOTAL"[0] := "DATOS AUXILIARES"."CONTADOR PVP TOTAL"[0] - 3.95;
       "DATOS AUXILIARES"."CONTADOR FACTURA TOTAL"[0] := "DATOS AUXILIARES"."CONTADOR FACTURA TOTAL"[0] - 3.95;
   END_IF;
END_REGION

REGION Network 2: RESTAR CAMELL
   RUNG wire#powerrail
      Contact( #RECTIFCAR )
      Contact( "DATOS AUXILIARES".DATOS[5] )
      Contact( "Tag_2" )
      P_Trig( "DATOS AUXILIARES".DATOS[25] )
      wire#w1
      { S7_Templates := "SrcType := Int"; S7_GenerateENO := "TRUE" } Sub(in1 := "DATOS AUXILIARES"."CONTADOR UNID."[1], in2 := 1, out => "DATOS AUXILIARES"."CONTADOR UNID."[1])
   END_RUNG
   RUNG wire#w1
      { S7_Templates := "SrcType := Real"; S7_GenerateENO := "TRUE" } Sub(in1 := "DATOS AUXILIARES"."CONTADOR PVP TOTAL"[1], in2 := 4.25, out => "DATOS AUXILIARES"."CONTADOR PVP TOTAL"[1])
   END_RUNG
   RUNG wire#w1
      { S7_Templates := "SrcType := Real"; S7_GenerateENO := "TRUE" } Sub(in1 := "DATOS AUXILIARES"."CONTADOR FACTURA TOTAL"[0], in2 := 4.25, out => "DATOS AUXILIARES"."CONTADOR FACTURA TOTAL"[0])
   END_RUNG
   // the same network as SCL:
   #_w1 := #RECTIFCAR AND "DATOS AUXILIARES".DATOS[5] AND "Tag_2";
   #_w2 := #_w1 AND NOT "DATOS AUXILIARES".DATOS[25];   // rising edge
   "DATOS AUXILIARES".DATOS[25] := #_w1;
   IF #_w2 THEN
       "DATOS AUXILIARES"."CONTADOR UNID."[1] := "DATOS AUXILIARES"."CONTADOR UNID."[1] - 1;
       "DATOS AUXILIARES"."CONTADOR PVP TOTAL"[1] := "DATOS AUXILIARES"."CONTADOR PVP TOTAL"[1] - 4.25;
       "DATOS AUXILIARES"."CONTADOR FACTURA TOTAL"[0] := "DATOS AUXILIARES"."CONTADOR FACTURA TOTAL"[0] - 4.25;
   END_IF;
END_REGION

REGION Network 3: RESTAR FORTUNA
   RUNG wire#powerrail
      Contact( #RECTIFCAR )
      Contact( "DATOS AUXILIARES".DATOS[9] )
      Contact( "Tag_2" )
      P_Trig( "DATOS AUXILIARES".DATOS[26] )
      wire#w1
      { S7_Templates := "SrcType := Int"; S7_GenerateENO := "TRUE" } Sub(in1 := "DATOS AUXILIARES"."CONTADOR UNID."[2], in2 := 1, out => "DATOS AUXILIARES"."CONTADOR UNID."[2])
   END_RUNG
   RUNG wire#w1
      { S7_Templates := "SrcType := Real"; S7_GenerateENO := "TRUE" } Sub(in1 := "DATOS AUXILIARES"."CONTADOR PVP TOTAL"[2], in2 := 4.35, out => "DATOS AUXILIARES"."CONTADOR PVP TOTAL"[2])
   END_RUNG
   RUNG wire#w1
      { S7_Templates := "SrcType := Real"; S7_GenerateENO := "TRUE" } Sub(in1 := "DATOS AUXILIARES"."CONTADOR FACTURA TOTAL"[0], in2 := 4.35, out => "DATOS AUXILIARES"."CONTADOR FACTURA TOTAL"[0])
   END_RUNG
   // the same network as SCL:
   #_w1 := #RECTIFCAR AND "DATOS AUXILIARES".DATOS[9] AND "Tag_2";
   #_w2 := #_w1 AND NOT "DATOS AUXILIARES".DATOS[26];   // rising edge
   "DATOS AUXILIARES".DATOS[26] := #_w1;
   IF #_w2 THEN
       "DATOS AUXILIARES"."CONTADOR UNID."[2] := "DATOS AUXILIARES"."CONTADOR UNID."[2] - 1;
       "DATOS AUXILIARES"."CONTADOR PVP TOTAL"[2] := "DATOS AUXILIARES"."CONTADOR PVP TOTAL"[2] - 4.35;
       "DATOS AUXILIARES"."CONTADOR FACTURA TOTAL"[0] := "DATOS AUXILIARES"."CONTADOR FACTURA TOTAL"[0] - 4.35;
   END_IF;
END_REGION

REGION Network 4: RESTAR LUCKY
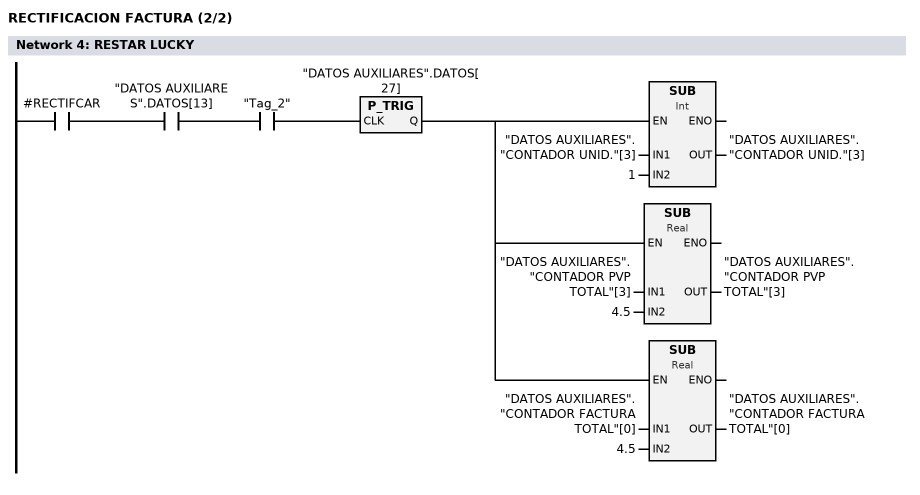
   RUNG wire#powerrail
      Contact( #RECTIFCAR )
      Contact( "DATOS AUXILIARES".DATOS[13] )
      Contact( "Tag_2" )
      P_Trig( "DATOS AUXILIARES".DATOS[27] )
      wire#w1
      { S7_Templates := "SrcType := Int"; S7_GenerateENO := "TRUE" } Sub(in1 := "DATOS AUXILIARES"."CONTADOR UNID."[3], in2 := 1, out => "DATOS AUXILIARES"."CONTADOR UNID."[3])
   END_RUNG
   RUNG wire#w1
      { S7_Templates := "SrcType := Real"; S7_GenerateENO := "TRUE" } Sub(in1 := "DATOS AUXILIARES"."CONTADOR PVP TOTAL"[3], in2 := 4.5, out => "DATOS AUXILIARES"."CONTADOR PVP TOTAL"[3])
   END_RUNG
   RUNG wire#w1
      { S7_Templates := "SrcType := Real"; S7_GenerateENO := "TRUE" } Sub(in1 := "DATOS AUXILIARES"."CONTADOR FACTURA TOTAL"[0], in2 := 4.5, out => "DATOS AUXILIARES"."CONTADOR FACTURA TOTAL"[0])
   END_RUNG
   // the same network as SCL:
   #_w1 := #RECTIFCAR AND "DATOS AUXILIARES".DATOS[13] AND "Tag_2";
   #_w2 := #_w1 AND NOT "DATOS AUXILIARES".DATOS[27];   // rising edge
   "DATOS AUXILIARES".DATOS[27] := #_w1;
   IF #_w2 THEN
       "DATOS AUXILIARES"."CONTADOR UNID."[3] := "DATOS AUXILIARES"."CONTADOR UNID."[3] - 1;
       "DATOS AUXILIARES"."CONTADOR PVP TOTAL"[3] := "DATOS AUXILIARES"."CONTADOR PVP TOTAL"[3] - 4.5;
       "DATOS AUXILIARES"."CONTADOR FACTURA TOTAL"[0] := "DATOS AUXILIARES"."CONTADOR FACTURA TOTAL"[0] - 4.5;
   END_IF;
END_REGION
END_FUNCTION

FUNCTION "CLASIFICADORA" : Void   // FC8, LAD
TITLE = CLASIFICADOR
{ S7_Optimized_Access := 'FALSE' }
VERSION : 0.1
// LOS PAQUETES SE DESPLAZAN POR UNA CINTA TRANSPORTADOR CENTRAL ,EL LECTOR  RECONOCE EL TIPO DE PRODUCTO Y CUANDO VAN PASANDO POR LOS SENSORES Y COINCIDE EL TIPO SE ACTIVA UN PISTON CON RETOCESO POR MUELLE QUE LOS DESPLAZA A OTRA CINTA INDEPENDIENTE PARA CADA PRODUCTO Y LOS DEPOSITA EN UN CONTENEDOR.SI EL LECTOR  NO ASOCIA EL CODIGO A NINGUN PRODUCTO SEGUIRA HASTA EL FINAL DE LA CINTA CENTRAL DONDE HAY UN CONTENEDOR PARA DESECHOS.
   VAR_INPUT
      "MARCHA CINTAS T." : Bool;
      "PARO CINTAS T." : Bool;
      "S1 PALL MALL" : Bool;
      "SC 1" : Bool;
      "S2 CAMELL" : Bool;
      "SC 2" : Bool;
      "S3 FORTUNA" : Bool;
      "SC 3" : Bool;
      "S4 LUCKY" : Bool;
      "SC 4" : Bool;
   END_VAR
   VAR_OUTPUT
      "P1 PALL MALL" : Bool;
      "P2 CAMELL" : Bool;
      "P3 FORTUNA" : Bool;
      "P4 LUCKY" : Bool;
      "CINTAS TRANSPOR.      CENTRAL,1,2,3,4" : Bool;
   END_VAR
   VAR_TEMP   // added for the SCL form of the ladder/FBD networks
      _w1 : Bool;
      _w2 : Bool;
   END_VAR
BEGIN

REGION Network 1: ARRANQUE CINTAS TRANSPORTADORAS(CENTRAL,1,2,3,4,)
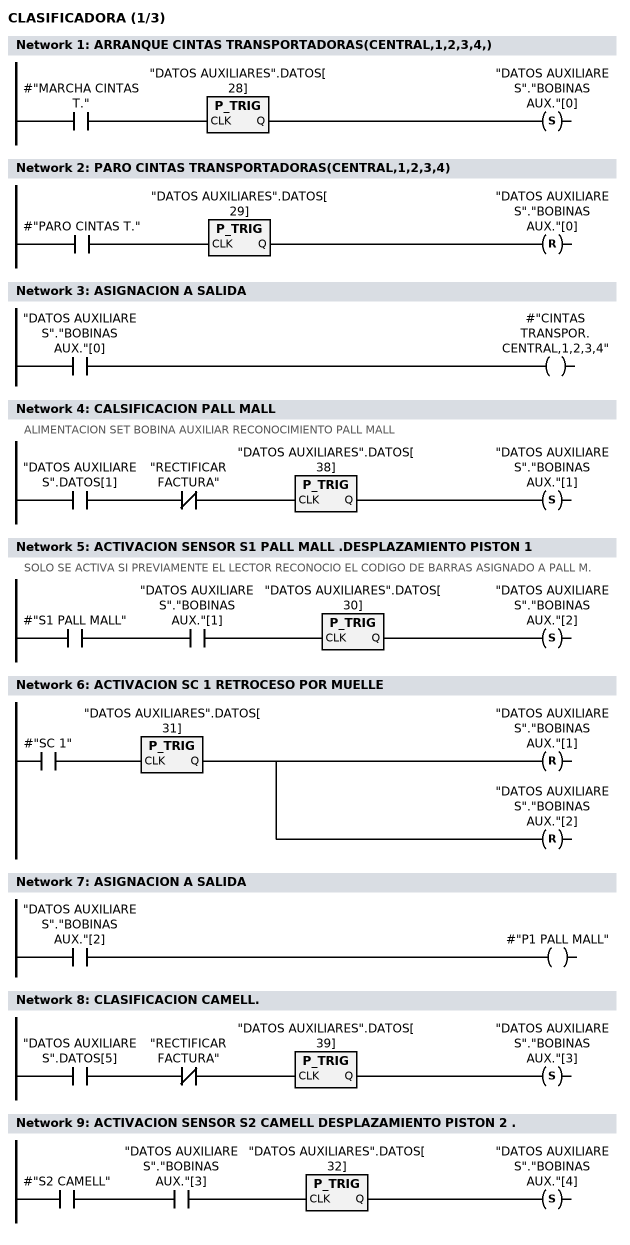
   RUNG wire#powerrail
      Contact( #"MARCHA CINTAS T." )
      P_Trig( "DATOS AUXILIARES".DATOS[28] )
      S_Coil( "DATOS AUXILIARES"."BOBINAS AUX."[0] )
   END_RUNG
   // the same network as SCL:
   #_w1 := #"MARCHA CINTAS T." AND NOT "DATOS AUXILIARES".DATOS[28];   // rising edge
   "DATOS AUXILIARES".DATOS[28] := #"MARCHA CINTAS T.";
   IF #_w1 THEN "DATOS AUXILIARES"."BOBINAS AUX."[0] := TRUE; END_IF;
END_REGION

REGION Network 2: PARO CINTAS TRANSPORTADORAS(CENTRAL,1,2,3,4)
   RUNG wire#powerrail
      Contact( #"PARO CINTAS T." )
      P_Trig( "DATOS AUXILIARES".DATOS[29] )
      R_Coil( "DATOS AUXILIARES"."BOBINAS AUX."[0] )
   END_RUNG
   // the same network as SCL:
   #_w1 := #"PARO CINTAS T." AND NOT "DATOS AUXILIARES".DATOS[29];   // rising edge
   "DATOS AUXILIARES".DATOS[29] := #"PARO CINTAS T.";
   IF #_w1 THEN "DATOS AUXILIARES"."BOBINAS AUX."[0] := FALSE; END_IF;
END_REGION

REGION Network 3: ASIGNACION A SALIDA
   RUNG wire#powerrail
      Contact( "DATOS AUXILIARES"."BOBINAS AUX."[0] )
      Coil( #"CINTAS TRANSPOR.      CENTRAL,1,2,3,4" )
   END_RUNG
   // the same network as SCL:
   #"CINTAS TRANSPOR.      CENTRAL,1,2,3,4" := "DATOS AUXILIARES"."BOBINAS AUX."[0];
END_REGION

REGION Network 4: CALSIFICACION PALL MALL
   // ALIMENTACION SET BOBINA AUXILIAR RECONOCIMIENTO PALL MALL
   RUNG wire#powerrail
      Contact( "DATOS AUXILIARES".DATOS[1] )
      I_Contact( "RECTIFICAR FACTURA" )
      P_Trig( "DATOS AUXILIARES".DATOS[38] )
      S_Coil( "DATOS AUXILIARES"."BOBINAS AUX."[1] )
   END_RUNG
   // the same network as SCL:
   #_w1 := "DATOS AUXILIARES".DATOS[1] AND NOT "RECTIFICAR FACTURA";
   #_w2 := #_w1 AND NOT "DATOS AUXILIARES".DATOS[38];   // rising edge
   "DATOS AUXILIARES".DATOS[38] := #_w1;
   IF #_w2 THEN "DATOS AUXILIARES"."BOBINAS AUX."[1] := TRUE; END_IF;
END_REGION

REGION Network 5: ACTIVACION SENSOR S1 PALL MALL .DESPLAZAMIENTO PISTON 1
   // SOLO SE ACTIVA SI PREVIAMENTE EL LECTOR RECONOCIO EL CODIGO DE BARRAS ASIGNADO A PALL M.
   RUNG wire#powerrail
      Contact( #"S1 PALL MALL" )
      Contact( "DATOS AUXILIARES"."BOBINAS AUX."[1] )
      P_Trig( "DATOS AUXILIARES".DATOS[30] )
      S_Coil( "DATOS AUXILIARES"."BOBINAS AUX."[2] )
   END_RUNG
   // the same network as SCL:
   #_w1 := #"S1 PALL MALL" AND "DATOS AUXILIARES"."BOBINAS AUX."[1];
   #_w2 := #_w1 AND NOT "DATOS AUXILIARES".DATOS[30];   // rising edge
   "DATOS AUXILIARES".DATOS[30] := #_w1;
   IF #_w2 THEN "DATOS AUXILIARES"."BOBINAS AUX."[2] := TRUE; END_IF;
END_REGION

REGION Network 6: ACTIVACION SC 1 RETROCESO POR MUELLE
   RUNG wire#powerrail
      Contact( #"SC 1" )
      P_Trig( "DATOS AUXILIARES".DATOS[31] )
      wire#w1
      R_Coil( "DATOS AUXILIARES"."BOBINAS AUX."[1] )
   END_RUNG
   RUNG wire#w1
      R_Coil( "DATOS AUXILIARES"."BOBINAS AUX."[2] )
   END_RUNG
   // the same network as SCL:
   #_w1 := #"SC 1" AND NOT "DATOS AUXILIARES".DATOS[31];   // rising edge
   "DATOS AUXILIARES".DATOS[31] := #"SC 1";
   IF #_w1 THEN
       "DATOS AUXILIARES"."BOBINAS AUX."[1] := FALSE;
       "DATOS AUXILIARES"."BOBINAS AUX."[2] := FALSE;
   END_IF;
END_REGION

REGION Network 7: ASIGNACION A SALIDA
   RUNG wire#powerrail
      Contact( "DATOS AUXILIARES"."BOBINAS AUX."[2] )
      Coil( #"P1 PALL MALL" )
   END_RUNG
   // the same network as SCL:
   #"P1 PALL MALL" := "DATOS AUXILIARES"."BOBINAS AUX."[2];
END_REGION

REGION Network 8: CLASIFICACION CAMELL.
   RUNG wire#powerrail
      Contact( "DATOS AUXILIARES".DATOS[5] )
      I_Contact( "RECTIFICAR FACTURA" )
      P_Trig( "DATOS AUXILIARES".DATOS[39] )
      S_Coil( "DATOS AUXILIARES"."BOBINAS AUX."[3] )
   END_RUNG
   // the same network as SCL:
   #_w1 := "DATOS AUXILIARES".DATOS[5] AND NOT "RECTIFICAR FACTURA";
   #_w2 := #_w1 AND NOT "DATOS AUXILIARES".DATOS[39];   // rising edge
   "DATOS AUXILIARES".DATOS[39] := #_w1;
   IF #_w2 THEN "DATOS AUXILIARES"."BOBINAS AUX."[3] := TRUE; END_IF;
END_REGION

REGION Network 9: ACTIVACION SENSOR S2 CAMELL DESPLAZAMIENTO PISTON 2 .
   RUNG wire#powerrail
      Contact( #"S2 CAMELL" )
      Contact( "DATOS AUXILIARES"."BOBINAS AUX."[3] )
      P_Trig( "DATOS AUXILIARES".DATOS[32] )
      S_Coil( "DATOS AUXILIARES"."BOBINAS AUX."[4] )
   END_RUNG
   // the same network as SCL:
   #_w1 := #"S2 CAMELL" AND "DATOS AUXILIARES"."BOBINAS AUX."[3];
   #_w2 := #_w1 AND NOT "DATOS AUXILIARES".DATOS[32];   // rising edge
   "DATOS AUXILIARES".DATOS[32] := #_w1;
   IF #_w2 THEN "DATOS AUXILIARES"."BOBINAS AUX."[4] := TRUE; END_IF;
END_REGION

REGION Network 10: ACTIVACION SC 2 RETROCESO POR MUELLE.....
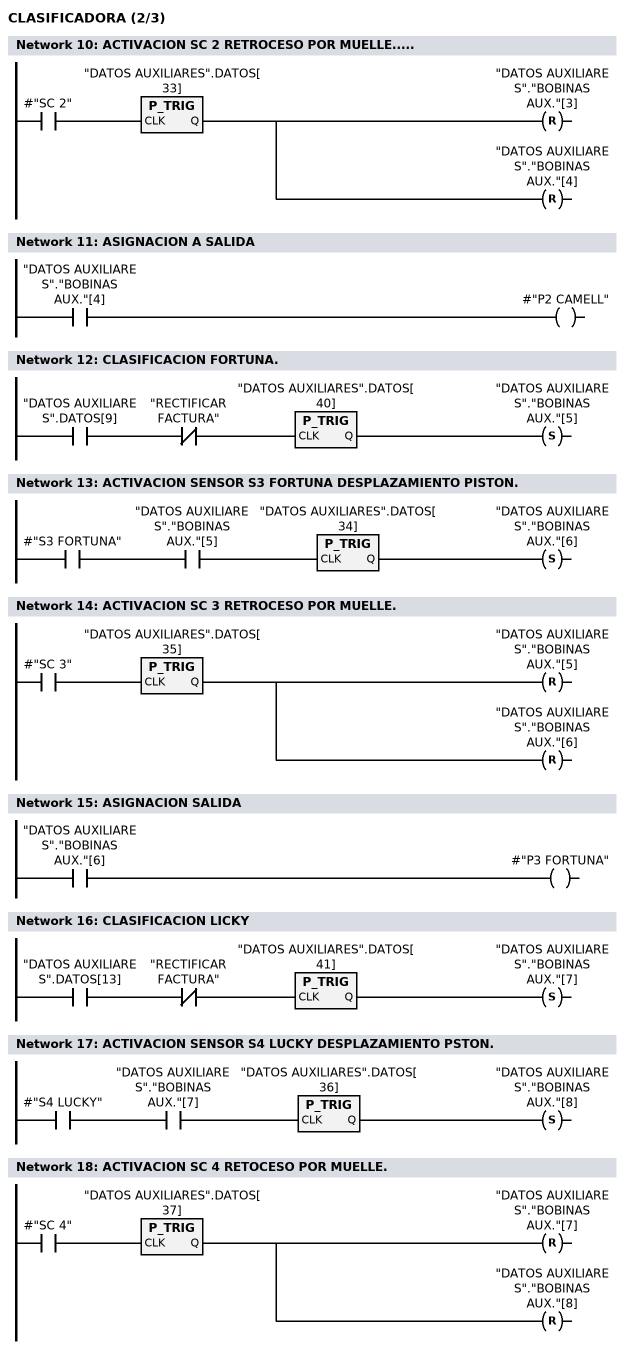
   RUNG wire#powerrail
      Contact( #"SC 2" )
      P_Trig( "DATOS AUXILIARES".DATOS[33] )
      wire#w1
      R_Coil( "DATOS AUXILIARES"."BOBINAS AUX."[3] )
   END_RUNG
   RUNG wire#w1
      R_Coil( "DATOS AUXILIARES"."BOBINAS AUX."[4] )
   END_RUNG
   // the same network as SCL:
   #_w1 := #"SC 2" AND NOT "DATOS AUXILIARES".DATOS[33];   // rising edge
   "DATOS AUXILIARES".DATOS[33] := #"SC 2";
   IF #_w1 THEN
       "DATOS AUXILIARES"."BOBINAS AUX."[3] := FALSE;
       "DATOS AUXILIARES"."BOBINAS AUX."[4] := FALSE;
   END_IF;
END_REGION

REGION Network 11: ASIGNACION A SALIDA
   RUNG wire#powerrail
      Contact( "DATOS AUXILIARES"."BOBINAS AUX."[4] )
      Coil( #"P2 CAMELL" )
   END_RUNG
   // the same network as SCL:
   #"P2 CAMELL" := "DATOS AUXILIARES"."BOBINAS AUX."[4];
END_REGION

REGION Network 12: CLASIFICACION FORTUNA.
   RUNG wire#powerrail
      Contact( "DATOS AUXILIARES".DATOS[9] )
      I_Contact( "RECTIFICAR FACTURA" )
      P_Trig( "DATOS AUXILIARES".DATOS[40] )
      S_Coil( "DATOS AUXILIARES"."BOBINAS AUX."[5] )
   END_RUNG
   // the same network as SCL:
   #_w1 := "DATOS AUXILIARES".DATOS[9] AND NOT "RECTIFICAR FACTURA";
   #_w2 := #_w1 AND NOT "DATOS AUXILIARES".DATOS[40];   // rising edge
   "DATOS AUXILIARES".DATOS[40] := #_w1;
   IF #_w2 THEN "DATOS AUXILIARES"."BOBINAS AUX."[5] := TRUE; END_IF;
END_REGION

REGION Network 13: ACTIVACION SENSOR S3 FORTUNA DESPLAZAMIENTO PISTON.
   RUNG wire#powerrail
      Contact( #"S3 FORTUNA" )
      Contact( "DATOS AUXILIARES"."BOBINAS AUX."[5] )
      P_Trig( "DATOS AUXILIARES".DATOS[34] )
      S_Coil( "DATOS AUXILIARES"."BOBINAS AUX."[6] )
   END_RUNG
   // the same network as SCL:
   #_w1 := #"S3 FORTUNA" AND "DATOS AUXILIARES"."BOBINAS AUX."[5];
   #_w2 := #_w1 AND NOT "DATOS AUXILIARES".DATOS[34];   // rising edge
   "DATOS AUXILIARES".DATOS[34] := #_w1;
   IF #_w2 THEN "DATOS AUXILIARES"."BOBINAS AUX."[6] := TRUE; END_IF;
END_REGION

REGION Network 14: ACTIVACION SC 3 RETROCESO POR MUELLE.
   RUNG wire#powerrail
      Contact( #"SC 3" )
      P_Trig( "DATOS AUXILIARES".DATOS[35] )
      wire#w1
      R_Coil( "DATOS AUXILIARES"."BOBINAS AUX."[5] )
   END_RUNG
   RUNG wire#w1
      R_Coil( "DATOS AUXILIARES"."BOBINAS AUX."[6] )
   END_RUNG
   // the same network as SCL:
   #_w1 := #"SC 3" AND NOT "DATOS AUXILIARES".DATOS[35];   // rising edge
   "DATOS AUXILIARES".DATOS[35] := #"SC 3";
   IF #_w1 THEN
       "DATOS AUXILIARES"."BOBINAS AUX."[5] := FALSE;
       "DATOS AUXILIARES"."BOBINAS AUX."[6] := FALSE;
   END_IF;
END_REGION

REGION Network 15: ASIGNACION SALIDA
   RUNG wire#powerrail
      Contact( "DATOS AUXILIARES"."BOBINAS AUX."[6] )
      Coil( #"P3 FORTUNA" )
   END_RUNG
   // the same network as SCL:
   #"P3 FORTUNA" := "DATOS AUXILIARES"."BOBINAS AUX."[6];
END_REGION

REGION Network 16: CLASIFICACION LICKY
   RUNG wire#powerrail
      Contact( "DATOS AUXILIARES".DATOS[13] )
      I_Contact( "RECTIFICAR FACTURA" )
      P_Trig( "DATOS AUXILIARES".DATOS[41] )
      S_Coil( "DATOS AUXILIARES"."BOBINAS AUX."[7] )
   END_RUNG
   // the same network as SCL:
   #_w1 := "DATOS AUXILIARES".DATOS[13] AND NOT "RECTIFICAR FACTURA";
   #_w2 := #_w1 AND NOT "DATOS AUXILIARES".DATOS[41];   // rising edge
   "DATOS AUXILIARES".DATOS[41] := #_w1;
   IF #_w2 THEN "DATOS AUXILIARES"."BOBINAS AUX."[7] := TRUE; END_IF;
END_REGION

REGION Network 17: ACTIVACION SENSOR S4 LUCKY DESPLAZAMIENTO PSTON.
   RUNG wire#powerrail
      Contact( #"S4 LUCKY" )
      Contact( "DATOS AUXILIARES"."BOBINAS AUX."[7] )
      P_Trig( "DATOS AUXILIARES".DATOS[36] )
      S_Coil( "DATOS AUXILIARES"."BOBINAS AUX."[8] )
   END_RUNG
   // the same network as SCL:
   #_w1 := #"S4 LUCKY" AND "DATOS AUXILIARES"."BOBINAS AUX."[7];
   #_w2 := #_w1 AND NOT "DATOS AUXILIARES".DATOS[36];   // rising edge
   "DATOS AUXILIARES".DATOS[36] := #_w1;
   IF #_w2 THEN "DATOS AUXILIARES"."BOBINAS AUX."[8] := TRUE; END_IF;
END_REGION

REGION Network 18: ACTIVACION SC 4 RETOCESO POR MUELLE.
   RUNG wire#powerrail
      Contact( #"SC 4" )
      P_Trig( "DATOS AUXILIARES".DATOS[37] )
      wire#w1
      R_Coil( "DATOS AUXILIARES"."BOBINAS AUX."[7] )
   END_RUNG
   RUNG wire#w1
      R_Coil( "DATOS AUXILIARES"."BOBINAS AUX."[8] )
   END_RUNG
   // the same network as SCL:
   #_w1 := #"SC 4" AND NOT "DATOS AUXILIARES".DATOS[37];   // rising edge
   "DATOS AUXILIARES".DATOS[37] := #"SC 4";
   IF #_w1 THEN
       "DATOS AUXILIARES"."BOBINAS AUX."[7] := FALSE;
       "DATOS AUXILIARES"."BOBINAS AUX."[8] := FALSE;
   END_IF;
END_REGION

REGION Network 19: ASIGNACION SALIDA
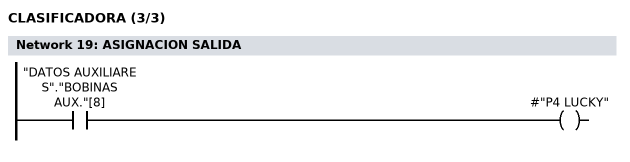
   RUNG wire#powerrail
      Contact( "DATOS AUXILIARES"."BOBINAS AUX."[8] )
      Coil( #"P4 LUCKY" )
   END_RUNG
   // the same network as SCL:
   #"P4 LUCKY" := "DATOS AUXILIARES"."BOBINAS AUX."[8];
END_REGION
END_FUNCTION

ORGANIZATION_BLOCK "Main"   // OB1, LAD
TITLE = LECTOR DE CODIGO DE BARRA TABACALERA. / "Main Program Sweep (Cycle)"
{ S7_Optimized_Access := 'FALSE' }
VERSION : 0.1
   VAR_TEMP
      OB1_EV_CLASS : Byte;   // Bits 0-3 = 1 (Coming event), Bits 4-7 = 1 (Event class 1)
      OB1_SCAN_1 : Byte;   // 1 (Cold restart scan 1 of OB 1), 3 (Scan 2-n of OB 1)
      OB1_PRIORITY : Byte;   // Priority of OB Execution
      OB1_OB_NUMBR : Byte;   // 1 (Organization block 1, OB1)
      OB1_RESERVED_1 : Byte;   // Reserved for system
      OB1_RESERVED_2 : Byte;   // Reserved for system
      OB1_PREV_CYCLE : Int;   // Cycle time of previous OB1 scan (milliseconds)
      OB1_MIN_CYCLE : Int;   // Minimum cycle time of OB1 (milliseconds)
      OB1_MAX_CYCLE : Int;   // Maximum cycle time of OB1 (milliseconds)
      OB1_DATE_TIME : Date_And_Time;   // Date and time OB1 started
   END_VAR
BEGIN
END_ORGANIZATION_BLOCK